// TIA Portal V17 export
// export: Created 2024-08-07T21:44:03.3644308Z, ExportSetting WithDefaults, DisplayName Totally Integrated Automation Portal, DisplayVersion V17 Update 7, DisplayName TIA Portal Openness, DisplayVersion V17 Update 7, DisplayName TIA Portal Version Control Interface, DisplayVersion V17, DisplayName SINAMICS Startdrive Advanced, DisplayVersion V17 SP2, DisplayName SINAMICS Startdrive G110M, G120, G120C, G120D, G120P, G115D, DisplayVersion V17 SP2, DisplayName SINAMICS Startdrive G130, G150, S120, S150, SINAMICS MV, S210, DisplayVersion V17 SP2, DisplayName STEP 7 Professional, DisplayVersion V17 Update 7, DisplayName STEP 7 Safety, DisplayVersion V17 Update 6, DisplayName WinCC Advanced / Unified PC, DisplayVersion V17 Update 7
DATA_BLOCK "PartErrorsCounter"   // DB46
{ S7_Optimized_Access := 'TRUE' }
VERSION : 0.1
// stored: AutoNumber true, DBAccessibleFromOPCUA true, DBAccessibleFromWebserver true, IsOnlyStoredInLoadMemory false, IsRetainMemResEnabled false, IsWriteProtectedInAS false, MemoryReserve 100
   VAR RETAIN
      CountersRef { S7_SetPoint := 'True'} : Array[1.."NumberOfProductionPrograms"] of "UDT_NOKcounter";
   END_VAR
   VAR
      CountersHMI : "UDT_NOKcounter";
   END_VAR
BEGIN
   CountersRef[1].Counters[0,0..50] := 0;
   CountersRef[1].Counters[1,0..9] := 0;
   CountersRef[1].Counters[1,10] := 2;
   CountersRef[1].Counters[1,11] := 1;
   CountersRef[1].Counters[1,12..19] := 0;
   CountersRef[1].Counters[1,20] := 3;
   CountersRef[1].Counters[1,21] := 1;
   CountersRef[1].Counters[1,22..33] := 0;
   CountersRef[1].Counters[1,34] := 1;
   CountersRef[1].Counters[1,35..43] := 0;
   CountersRef[1].Counters[1,44] := 1;
   CountersRef[1].Counters[1,45..50] := 0;
   CountersRef[1].Counters[2,0..13] := 0;
   CountersRef[1].Counters[2,14] := 1;
   CountersRef[1].Counters[2,15..20] := 0;
   CountersRef[1].Counters[2,21] := 1;
   CountersRef[1].Counters[2,22..50] := 0;
   CountersRef[1].Counters[3,0..50] := 0;
   CountersRef[2].Counters[0,0..50] := 0;
   CountersRef[2].Counters[1,0..9] := 0;
   CountersRef[2].Counters[1,10] := 4;
   CountersRef[2].Counters[1,11] := 1;
   CountersRef[2].Counters[1,12..19] := 0;
   CountersRef[2].Counters[1,20] := 3;
   CountersRef[2].Counters[1,21] := 2;
   CountersRef[2].Counters[1,22..50] := 0;
   CountersRef[2].Counters[2,0..10] := 0;
   CountersRef[2].Counters[2,11] := 1;
   CountersRef[2].Counters[2,12..13] := 0;
   CountersRef[2].Counters[2,14] := 1;
   CountersRef[2].Counters[2,15..20] := 0;
   CountersRef[2].Counters[2,21] := 1;
   CountersRef[2].Counters[2,22..23] := 0;
   CountersRef[2].Counters[2,24] := 1;
   CountersRef[2].Counters[2,25..30] := 0;
   CountersRef[2].Counters[2,31] := 1;
   CountersRef[2].Counters[2,32..33] := 0;
   CountersRef[2].Counters[2,34] := 1;
   CountersRef[2].Counters[2,35..40] := 0;
   CountersRef[2].Counters[2,41] := 1;
   CountersRef[2].Counters[2,42..43] := 0;
   CountersRef[2].Counters[2,44] := 1;
   CountersRef[2].Counters[2,45..50] := 0;
   CountersRef[2].Counters[3,0..50] := 0;
   CountersRef[3].Counters[0,0..50] := 0;
   CountersRef[3].Counters[1,0..50] := 0;
   CountersRef[3].Counters[2,0..50] := 0;
   CountersRef[3].Counters[3,0..50] := 0;
   CountersRef[4].Counters[0,0..50] := 0;
   CountersRef[4].Counters[1,0..50] := 0;
   CountersRef[4].Counters[2,0..50] := 0;
   CountersRef[4].Counters[3,0..50] := 0;
   CountersRef[5].Counters[0,0..50] := 0;
   CountersRef[5].Counters[1,0..9] := 0;
   CountersRef[5].Counters[1,10] := 17;
   CountersRef[5].Counters[1,11] := 6;
   CountersRef[5].Counters[1,12..19] := 0;
   CountersRef[5].Counters[1,20..21] := 1;
   CountersRef[5].Counters[1,22..50] := 0;
   CountersRef[5].Counters[2,0..9] := 0;
   CountersRef[5].Counters[2,10] := 4;
   CountersRef[5].Counters[2,11] := 3;
   CountersRef[5].Counters[2,12..13] := 0;
   CountersRef[5].Counters[2,14] := 1;
   CountersRef[5].Counters[2,15..23] := 0;
   CountersRef[5].Counters[2,24] := 4;
   CountersRef[5].Counters[2,25..50] := 0;
   CountersRef[5].Counters[3,0..50] := 0;
   CountersRef[6].Counters[0,0..50] := 0;
   CountersRef[6].Counters[1,0..50] := 0;
   CountersRef[6].Counters[2,0..9] := 0;
   CountersRef[6].Counters[2,10] := 1;
   CountersRef[6].Counters[2,11..13] := 0;
   CountersRef[6].Counters[2,14] := 1;
   CountersRef[6].Counters[2,15..21] := 0;
   CountersRef[6].Counters[2,22] := 1;
   CountersRef[6].Counters[2,23..33] := 0;
   CountersRef[6].Counters[2,34] := 2;
   CountersRef[6].Counters[2,35..43] := 0;
   CountersRef[6].Counters[2,44] := 2;
   CountersRef[6].Counters[2,45..50] := 0;
   CountersRef[6].Counters[3,0..50] := 0;
   CountersRef[7].Counters[0,0..50] := 0;
   CountersRef[7].Counters[1,0..50] := 0;
   CountersRef[7].Counters[2,0..50] := 0;
   CountersRef[7].Counters[3,0..50] := 0;
   CountersRef[8].Counters[0,0..50] := 0;
   CountersRef[8].Counters[1,0..50] := 0;
   CountersRef[8].Counters[2,0..50] := 0;
   CountersRef[8].Counters[3,0..50] := 0;
   CountersHMI.Counters[0,0..50] := 0;
   CountersHMI.Counters[1,0..50] := 0;
   CountersHMI.Counters[2,0..50] := 0;
   CountersHMI.Counters[3,0..50] := 0;
END_DATA_BLOCK
